DATA_BLOCK "CalcVolume_Tank10_DB"
{ S7_Optimized_Access := 'FALSE' }
VERSION : 0.1
"CalculationVolume"

BEGIN
   IW_Radius := 1.468;
   IW_ValueFromSensor := 18.56192;
   IW_K_for_Tonnag := 1.35;
   IW_K_for_Level := 1.35;
   QW_Volume := 93.04028;
   QW_Tonnag := 125.6044;
   QW_RealLevel := 13.74957;
   sW_S := 6.766776;
   sW_Volume := 93.04028;
   sW_RealLevel := 13.74957;

END_DATA_BLOCK

